# B&R Automation Studio project Tmp_Explorer_V1
Automation Studio 6.7.1.4; technology packages: mappServices 6.7.1, mappView 6.7.0, OpcUaCs 6.7.0

## Configuration X20CPU

CPU X20CP3687X, AutomationRuntime 6.7.8, Build 11.3.0, Safety 0.0

### Task classes (Cpu.sw)
```
Cyclic#8:
  FileExplor <- mappFileExplorer.FileExplorer.prg
  UsbDevice <- USBdevice.UsbDevice.prg
  NetDevice <- NETdevice.NetDevice.prg
Binaries: udbdef, mvLoader, TCData, ArSvcReg, mvConfig, arconfig, User, Role, iomap, asfw, ashwac, ashwd, sysconf, UaCsConfig, BRRole, Config, OpcUaMap
Libraries: FileIO, runtime, AsBrStr, AsUSB, standard, IecCheck, sys_lib, AsZip, AsICMP, astime, asieccon, UaCoalPrv, ArSsl, UaCoal, UaCore, MpServer, MpFile, MpBase
```

### Hardware
```
X20CP3687X : X20CP3687X v1.9.0.0
  Connector IF2:
    ActivateDevice = 1
    ActivateSnmp = 2
  Connector IF3:
    DNAConfiguration = manual
    CycleTime = 2000
  ConfigurationID = Tmp_Explorer_V1_X20CPU
  UserPartitionSize = 200
  VolatileGlobalPvSize = 200000
  EnableDebugger = 1
  FileDevice1
  FileDeviceName1 = USER
  FileDevicePath1 = USER_PATH
  ActivateFtpServer = 1
  FtpUser1
  FtpUsername1 = admin
  FtpUserPassword1 = 63faJ9mPKpD1G9ieIVwnNiGLd8KDZIbzebN9VYfcRfQ=  // admin
  FtpUserSalt1 = HY8+Pzqd
  FTPAccessRight1 = 0
  ActivateWebServer = 1
  ActivateSdm = 1
```

### Config.mpfilemanager - X20CP3687X/mappServices/Config.mpfilemanager
```
Element FileManagement (Type=mpfilemanager)
  mapp.Gen:
    Enable = TRUE
    EnableCockpit = TRUE
    Audit = TRUE
    Parent
  FileManager:
    USB = 0
    Devices:
      0:
        DeviceName = USER
        Text = USER
    Access:
      0:
        Folder = *
        Roles:
          0:
            Role = Everyone
            Rights:
              Visible = TRUE
              FolderRead = TRUE
              FileRead = TRUE
              FileEdit = TRUE
              FolderEdit = TRUE
          1:
            Role = Administrator
            Rights:
              Visible = TRUE
              FolderRead = TRUE
              FileRead = TRUE
              FileEdit = TRUE
              FolderEdit = TRUE
```

## Logical view

Binary libraries used (declarations not repeated): operator, runtime, astime, AsIecCon, FileIO, AsBrStr, AsUSB, standard, IecCheck, sys_lib, AsZip, AsICMP, MpServer 6.7.0, MpFile 6.7.1, MpBase

### compile_flags.txt
```
# This file is auto-generated by ASX. Do not edit manually, as changes may be overwritten.
# If you need to manually edit this file and prevent automatic updates, add "# MANUAL EDIT" to the first line.
-I
C:\Program Files (x86)\BrAutomation\AS6\AS\gnuinst\V11.3.0\6.0\i686-elf\include\c++\11.3.0
-I
C:\Program Files (x86)\BrAutomation\AS6\AS\gnuinst\V11.3.0\6.0\i686-elf\include\c++\11.3.0\i686-elf
-I
C:\Program Files (x86)\BrAutomation\AS6\AS\gnuinst\V11.3.0\6.0\i686-elf\include\c++\11.3.0\backward
-I
C:\Program Files (x86)\BrAutomation\AS6\AS\gnuinst\V11.3.0\6.0\lib\gcc\i686-elf\11.3.0\include
-I
C:\Program Files (x86)\BrAutomation\AS6\AS\gnuinst\V11.3.0\6.0\lib\gcc\i686-elf\11.3.0\include-fixed
-I
C:\Program Files (x86)\BrAutomation\AS6\AS\gnuinst\V11.3.0\6.0\i686-elf\include
-I
c:\Projects\Samples\mapp\mappExplorer\Temp\Includes
-trigraphs
-fno-asm
-D
_DEFAULT_INCLUDES
-D
_SG4
--target=i686-elf
-fPIC
-Wall
```

### ExplorerTypes.typ
```iecst
TYPE
	ClientInfoType : 	STRUCT
		userId : WSTRING[80];
		isValid : BOOL;
		ipAddress : WSTRING[15];
		languageId : WSTRING[2];
		screenResolution : WSTRING[32];
		slotId : SINT;
	END_STRUCT;
	expSTATE :
		( (*Explorer state machine*)
		EXP_WAIT,
		EXP_READ_DIR,
		EXP_READ_DIR_1,
		EXP_READ_DIR_2,
		EXP_READ_DIR_3,
		EXP_READ_DIR_4,
		EXP_DIR_CHANGE,
		EXP_COPY_ALL,
		EXP_FILE_COPY,
		EXP_FILE_DELETE,
		EXP_FILE_RENAME,
		EXP_FILE_DUPLICATE,
		EXP_FILE_VIEW,
		EXP_FILE_DOWNLOAD,
		EXP_FILE_DOWNLOAD_1,
		EXP_FILE_DOWNLOAD_DIR,
		EXP_FILE_UPLOAD,
		EXP_FILE_UPLOAD_1,
		EXP_DIR_COPY,
		EXP_DIR_CREATE,
		EXP_DIR_DELETE,
		EXP_DIR_RENAME,
		EXP_OVERWRITE_1,
		EXP_OVERWRITE_2
		);
	expERR : 	STRUCT  (*Sub structure error*)
		text : STRING[150]; (* Error text *)
		state : expSTATE; (* Error step *)
	END_STRUCT;
	expCMD : 	STRUCT  (*Sub structure commands*)
		refresh : BOOL; (*Read directory and file names from devices *)
		dir_change : BOOL; (*Change current directory *)
		dir_create : BOOL; (*Create a new directory *)
		copy : BOOL; (*Copy selected item from device a TO device b *)
		copy_all : BOOL; (*Copy all items from device a TO device b	*)
		view_file : BOOL; (*View selected file in mappView*)
		delete : BOOL; (*Delete selected file *)
		rename : BOOL; (*Rename selected file*)
		duplicate : BOOL; (*Duplicate selected file*)
		download : BOOL; (*Download selected file*)
		upload : BOOL; (*Upload file to target*)
	END_STRUCT;
	expPAR : 	STRUCT  (*Sub structure parameters*)
		device_active : STRING[40]; (*Active device name *)
		device_list : ARRAY[0..6]OF STRING[40]; (*List of all devices*)
		item_filter : STRING[EXPL_ITEM_LENGTH]; (*Only show files with this extension	*)
		new_name : STRING[EXPL_ITEM_LENGTH]; (*Name for for directory create and rename*)
		dir_path : STRING[EXPL_DIR_PATH_LENGTH]; (*Current directory path	*)
	END_STRUCT;
	expDAT : 	STRUCT  (*Sub structure data*)
		item_list : ARRAY[0..EXPL_LIST_NUM]OF STRING[EXPL_ITEM_LENGTH]; (*List with file names	*)
		item_size : ARRAY[0..EXPL_LIST_NUM]OF STRING[EXPL_SIZE_LENGTH]; (*List with file sizes*)
		item_num : UINT; (*Number of files	 displayed*)
		device_free : UINT; (*Free memory on device in MB*)
		device_size : UINT; (*Total memory size of device in MB*)
	END_STRUCT;
	expVIS : 	STRUCT  (*Sub structure visualization*)
		item_selected : UINT; (*Current selected file *)
		enable_button_set_1 : BOOL; (*Enable or disable buttons copy and delete*)
		enable_button_set_2 : BOOL; (*Enable or disable buttons refresh and create*)
		view_file_path : STRING[EXPL_DIR_PATH_LENGTH]; (*Full path for viewing file*)
		view_file : BOOL; (*Show message box on error*)
		download_execute : BOOL; (*Start downloading file*)
		file_status : DINT; (*Status of download and upload*)
		upload_execute : BOOL; (*Start uploading file*)
		file_full_path : STRING[EXPL_DIR_PATH_LENGTH]; (*File upload and download url*)
		overwrite_request : BOOL; (*Show message box to overwrite file*)
		overwrite_response : USINT; (*Response from message box overwrite file*)
		reload_upload : BOOL; (*Reload upload button*)
		double_click_event : USINT; (*Helper variable for double click in item list*)
		device_list : ARRAY[0..6]OF STRING[80]; (* Device name *)
	END_STRUCT;
	expMAIN : 	STRUCT  (*Main explorer structure*)
		CMD : ARRAY[0..1]OF expCMD; (* Command structure *)
		PAR : ARRAY[0..1]OF expPAR; (* Parameter structure *)
		DAT : ARRAY[0..1]OF expDAT; (*Data structure*)
		VIS : ARRAY[0..1]OF expVIS; (*Visualization structure*)
		ERR : expERR; (* Error structure *)
		status_no : DINT; (*Shows the status as number*)
		status_text : STRING[50]; (*Shows the status as text*)
	END_STRUCT;
END_TYPE
```

### ExplorerVariables.var
```iecst
VAR CONSTANT
	EXPL_DIR_PATH_LENGTH : UINT := 200; (*Maximum length for the complete path *)
	EXPL_LIST_NUM : UINT := 100; (*Maximum number if files and folders that can be listed *)
	EXPL_ITEM_LENGTH : USINT := 50; (*Maximum length for a file or folder name *)
	EXPL_SIZE_LENGTH : USINT := 15; (*Maximum length for a file or folder size*)
	EXPL_DEVICE_LIST : ARRAY[0..6] OF STRING[40] := ['USER','USB_DEVICE1','USB_DEVICE2','USB_DEVICE3','NET_DEVICE','','']; (*List of predefined devices *)
END_VAR
VAR
	EXPL_VIEW_FILTER : ARRAY[0..9] OF STRING[5] := ['csv','xml','txt','bmp','jpg',5('')]; (*Files extensions than can be used with the view command*)
	EXPL : expMAIN; (*Explorer main structure*)
END_VAR
```

### Program Logical/mappFileExplorer/FileExplorer (IEC)

#### Variables.var
```iecst
(*Local constants*)
VAR CONSTANT
	OK : USINT := 0; (*Status OK *)
	FILTER_AUTO_REFRESH : BOOL := TRUE; (*Auto refresh when filter changes *)
	COPY_AUTO_SELECT : USINT := 1; (*Select target item after copying *)
	COPY_AUTO_REFRESH : USINT := 1; (*Refresh items after copying *)
END_VAR
(*Local Variables*)
VAR
	side : BOOL := FALSE; (*Current side *)
	step : expSTATE := (0); (*Main step index *)
	animation : USINT := 0; (*Animation for working status	*)
	do_select : USINT := 0; (*Select item after copying *)
	old_filter : ARRAY[0..1] OF STRING[EXPL_ITEM_LENGTH]; (*Track filter change *)
	has_oversized_items : BOOL;
	tmp_str1 : STRING[EXPL_DIR_PATH_LENGTH]; (* Temporary STRING variable *)
	tmp_str2 : STRING[EXPL_DIR_PATH_LENGTH]; (* Temporary STRING variable *)
	tmp_str3 : STRING[EXPL_DIR_PATH_LENGTH]; (* Temporary STRING variable *)
	tmp_str4 : STRING[EXPL_DIR_PATH_LENGTH]; (* Temporary STRING variable *)
	lx : UDINT := 0; (* Index	*)
	ly : UINT;
	double_click_timer : TON_10ms;
	device_active_old : ARRAY[0..1] OF STRING[40];
	dir_path : STRING[EXPL_DIR_PATH_LENGTH];
	device_active : STRING[40];
	item_name : STRING[EXPL_DIR_PATH_LENGTH];
	duplicate_index : UDINT;
	duplicate_dot_pos : DINT;
	duplicate_suffix_pos : DINT;
	duplicate_suffix_valid : BOOL;
	duplicate_base_name : STRING[EXPL_ITEM_LENGTH];
	duplicate_extension : STRING[EXPL_ITEM_LENGTH];
	duplicate_suffix_text : STRING[EXPL_ITEM_LENGTH];
END_VAR
(*Local function calls*)
VAR
	DInfo : DirInfo;
	DOpen : DirOpen;
	DRead : DirReadEx;
	DClose : DirClose;
	FCopy : FileCopy;
	FDelete : FileDelete;
	FRename : FileRename;
	DCopy : DirCopy;
	DCreate : DirCreate;
	DDelete : DirDeleteEx;
	DRename : DirRename;
	DMemInfo : DevMemInfo;
	DevLink_0 : DevLink;
	lDirReadData : fiDIR_READ_EX_DATA;
	zipArchive_0 : zipArchive;
END_VAR
(*Local constants*)
VAR CONSTANT
	NONE : USINT := 0;
	YES : USINT := 1;
	NO : USINT := 2;
	ERR_EMPTY_ITEM : UINT := 50000; (*Selected item name is empty	*)
	ERR_INVALID_ITEM_NAME : UINT := 50001; (*This is not a valid item name*)
	ERR_DEVICE_UNDEFINED : UINT := 50010; (*Device is not defined*)
	ERR_MAX_FILES_REACHED : UINT := 50100; (*Maximum number of files reached*)
	ERR_NAME_EXCEEDS_MAX : UINT := 50200; (*File name exceeds maximum length*)
	ERR_DIR_EXCEEDS_MAX : UINT := 50201; (*Directory name exceeds maximum length*)
	ERR_PATH_EXCEEDS_MAX : UINT := 50202; (*Directory path exceeds maximum length*)
	ERR_PATH_CRITICAL : UINT := 50203; (*Directory path critical error*)
	ERR_PATH_RECURSIVE : UINT := 50204; (*Can not copy directory into itself*)
	ERR_DIR_DOWNLOAD_INVALID : UINT := 50331; (*This is not a valid directory for downloading*)
END_VAR
```

#### LocalFunctions.fun
```iecst
FUNCTION ReplaceString : BOOL
	VAR_INPUT
		dataSTR : UDINT;
		searchSTR : UDINT;
		replaceSTR : UDINT;
		first : BOOL;
	END_VAR
	VAR
		idx : UDINT;
	END_VAR
END_FUNCTION

FUNCTION IsInstr : BOOL
	VAR_INPUT
		string1 : UDINT;
		string2 : UDINT;
	END_VAR
	VAR
		idx : UDINT;
	END_VAR
END_FUNCTION

FUNCTION FindInMem : DINT
	VAR_INPUT
		data1 : UDINT;
		len1 : UDINT;
		data2 : UDINT;
		len2 : UDINT;
		direction : BOOL;
	END_VAR
	VAR
		idx : UDINT;
	END_VAR
END_FUNCTION

{REDUND_ERROR} FUNCTION CreateError : expSTATE (*TODO: Add your comment here*) (*$GROUP=User,$CAT=User,$GROUPICON=User.png,$CATICON=User.png*)
	VAR_INPUT
		nr : DINT;
		side : BOOL;
		step : expSTATE;
		text : STRING[150];
		EXPL : REFERENCE TO expMAIN;
	END_VAR
END_FUNCTION

FUNCTION InsertRecName : BOOL
	VAR_INPUT
		EXPL : REFERENCE TO expMAIN;
		new_name : STRING[EXPL_ITEM_LENGTH];
		size : STRING[15];
		side : BOOL;
	END_VAR
	VAR
		idx : DINT;
		idy : DINT;
		lSort : DINT;
	END_VAR
END_FUNCTION

FUNCTION WorkingStatus : USINT
	VAR_INPUT
		EXPL : REFERENCE TO expMAIN;
		str : UDINT;
		animation : USINT;
	END_VAR
END_FUNCTION

FUNCTION CreateCompletePath : BOOL
	VAR_INPUT
		path : STRING[EXPL_DIR_PATH_LENGTH];
		target : STRING[EXPL_ITEM_LENGTH];
		return_path : UDINT;
	END_VAR
	VAR
		tmp : STRING[EXPL_ITEM_LENGTH];
	END_VAR
END_FUNCTION

FUNCTION String2DataProvider : BOOL
	VAR_INPUT
		SourceString : UDINT;
		TargetString : UDINT;
	END_VAR
END_FUNCTION
```

#### LocalFunctions.st
```iecst
//******************************************************************************************************
// Create mappView data provider string
//******************************************************************************************************
FUNCTION String2DataProvider
	brsstrcpy(TargetString, ADR('{"value":"'));
	brsstrcat(TargetString, SourceString);
	brsstrcat(TargetString, ADR('","text":"'));
	brsstrcat(TargetString, SourceString);
	brsstrcat(TargetString, ADR('"}'));
	String2DataProvider := TRUE;
END_FUNCTION

//******************************************************************************************************
// Raise error function
//******************************************************************************************************
FUNCTION CreateError
	// Generate for known errors
	IF (nr = fiERR_NOT_ENOUGH_FREEMEM) THEN
		EXPL.ERR.text := 'not enough memory available on the target device';
	ELSIF (nr = fiERR_FILE_DEVICE) THEN
		EXPL.ERR.text := 'device is not connected';
	ELSIF (nr = fiERR_INVALID_PATH) THEN
		EXPL.ERR.text := 'directory is too long, does not exist or has invalid characters';
	ELSIF (nr = fiERR_DIR_NOT_EXIST) THEN
		EXPL.ERR.text := 'directory does not exist';
	ELSIF (nr = fiERR_FILE_DEVICE) THEN
		EXPL.ERR.text := 'directory path does not exist';
	ELSIF (nr = fiERR_DIR_ALREADY_EXIST) THEN
		EXPL.ERR.text := 'directory or file already exists';
	ELSIF (nr = fiERR_EXIST) THEN
		EXPL.ERR.text := 'directory or file already exists';
	ELSE
		EXPL.ERR.text := text;
	END_IF
	// Convert to error structure
	IF (side = 0) THEN
		brsstrcat(ADR(EXPL.ERR.text), ADR(' on side a'));
	ELSE
		brsstrcat(ADR(EXPL.ERR.text), ADR(' on side b'));
	END_IF
	EXPL.status_no 	:= nr;
	EXPL.ERR.state 	:= step;
	// When error occurs in dir read call dir close before reporting error
	IF (step = EXP_READ_DIR_2) THEN
		CreateError := EXP_READ_DIR_3;
	ELSE
		// Reset all commands
		brsmemset(ADR(EXPL.CMD[side]), 0, SIZEOF(EXPL.CMD[side]));
		brsmemset(ADR(EXPL.CMD[NOT side]), 0, SIZEOF(EXPL.CMD[NOT side]));
		CreateError := EXP_WAIT;
	END_IF
END_FUNCTION

//******************************************************************************************************
// Create complete path string
//******************************************************************************************************
FUNCTION CreateCompletePath
	brsmemset(ADR(tmp), 0, EXPL_ITEM_LENGTH);
	brsstrcpy(return_path, ADR(path));

	// ------------------------------------------------------------------------------------------------
	// Filter directory name
	IF(brsmemcmp(ADR(target), ADR('(DIR)'), 5) = 0) THEN
		brsmemcpy(ADR(tmp), ADR(target)+5, brsstrlen(ADR(target))-5);
	ELSE
		brsstrcpy(ADR(tmp), ADR(target));
	END_IF

	// ------------------------------------------------------------------------------------------------
	// Create directory path
	IF(path = '/') THEN
		brsstrcpy(return_path, ADR(tmp));
	ELSE
		brsstrcat(return_path, ADR('/'));
		brsstrcat(return_path, ADR(tmp));
	END_IF
	//	brsstrcat(return_path, ADR('/'));

	CreateCompletePath := FALSE;
END_FUNCTION

//******************************************************************************************************
// Working status
//******************************************************************************************************
FUNCTION WorkingStatus
	animation := animation+1;

	IF (animation = 80) THEN
		animation := 0;
	END_IF

	brsmemset(ADR(EXPL.status_text), 0, SIZEOF(EXPL.status_text));
	brsstrcpy(ADR(EXPL.status_text), str);
	CASE(animation) OF
		0..19	: brsstrcat(ADR(EXPL.status_text), ADR('/'));
		20..39	: brsstrcat(ADR(EXPL.status_text), ADR('-'));
		40..59	: brsstrcat(ADR(EXPL.status_text), ADR('\'));
		60..79	: brsstrcat(ADR(EXPL.status_text), ADR('|'));
	END_CASE;
	WorkingStatus := animation;
END_FUNCTION

//******************************************************************************************************
// Fill new folder or directory name
//******************************************************************************************************
FUNCTION InsertRecName
	// Set up start values for iteration
	IF (EXPL.DAT[side].item_num <> 0) THEN
		idy := EXPL.DAT[side].item_num - 1;
	END_IF
	idx := idy;

	// Start iteration	search
	WHILE (idy > 1) DO
		// Check current entry
		lSort := brsstrcmp(ADR(new_name), ADR(EXPL.DAT[side].item_list[idy]));
		// Solve new search range
		IF (idy MOD 2 = 0) THEN
			idy := idy / 2;
		ELSE
			idy := idy / 2 + 1;
		END_IF
		// New range is lower or higher than current
		IF (lSort > 0) THEN
			idx := idx + idy;
			IF (idx > UINT_TO_INT(EXPL.DAT[side].item_num)) THEN
				idx := EXPL.DAT[side].item_num;
			END_IF
		ELSE
			idx := idx - idy;
			IF (idx < 1) THEN
				idx := 1;
			END_IF
		END_IF
	END_WHILE;

	// New entry is this, next or previous
	lSort := brsstrcmp(ADR(new_name), ADR(EXPL.DAT[side].item_list[idx]));
	IF (lSort > 0 AND idx <> UINT_TO_INT(EXPL.DAT[side].item_num)) THEN
		idx := idx +1;
	ELSIF (idx > 0) THEN
		lSort := brsstrcmp(ADR(new_name), ADR(EXPL.DAT[side].item_list[idx-1]));
		IF (lSort < 0) THEN
			idx := idx - 1;
		END_IF
	END_IF

	// Force ".." at beginning of list
	IF (idx = 0 AND EXPL.DAT[side].item_list[0] = '..') THEN
		idx := idx + 1;
	END_IF
	// Move all data entrys backwards and fill in new entry
	IF(idx < EXPL_LIST_NUM) THEN
		brsmemmove(ADR(EXPL.DAT[side].item_list[idx+1]),ADR(EXPL.DAT[side].item_list[idx]), (EXPL.DAT[side].item_num - idx) * SIZEOF(EXPL.DAT[side].item_list[0]));
		brsmemmove(ADR(EXPL.DAT[side].item_size[idx+1]),ADR(EXPL.DAT[side].item_size[idx]), (EXPL.DAT[side].item_num - idx) * SIZEOF(EXPL.DAT[side].item_size[0]));
	END_IF
	brsstrcpy(ADR(EXPL.DAT[side].item_list[idx]), ADR(new_name));
	// Create data structure for vis size list
	brsstrcpy(ADR(EXPL.DAT[side].item_size[idx]), ADR(size));

	InsertRecName := TRUE;
END_FUNCTION

//******************************************************************************************************
// Is second string in first string
//******************************************************************************************************
FUNCTION IsInstr
	IF (brsstrlen(string1) > brsstrlen(string2)) THEN
		FOR idx:=0 TO brsstrlen(string1) - brsstrlen(string2) DO
			IF (brsmemcmp(string1 + idx, string2, brsstrlen(string2)) = 0) THEN
				IsInstr := TRUE;
				EXIT;
			END_IF
		END_FOR;
	END_IF
END_FUNCTION

//******************************************************************************************************
// Find second data in first data
//******************************************************************************************************
FUNCTION FindInMem
	FindInMem := -1;
	IF (len1 > len2) THEN
		IF(direction) THEN
			idx := len1 - len2;
			WHILE(idx > 0) DO
				IF (brsmemcmp(data1 + idx, data2, len2) = 0) THEN
					FindInMem := idx;
					EXIT;
				END_IF
				idx := idx - 1;
			END_WHILE;
		ELSE
			FOR idx:=0 TO len1 - len2 DO
				IF (brsmemcmp(data1 + idx, data2, len2) = 0) THEN
					FindInMem := idx;
					EXIT;
				END_IF
			END_FOR;
		END_IF
	END_IF
END_FUNCTION

//******************************************************************************************************
// Find and replace string
//******************************************************************************************************
FUNCTION ReplaceString
	IF (brsstrlen(dataSTR) >= brsstrlen(searchSTR)) THEN
		FOR idx:=0 TO brsstrlen(dataSTR) - brsstrlen(searchSTR) DO
			IF (brsmemcmp(dataSTR + idx, searchSTR, brsstrlen(searchSTR)) = 0) THEN
				// Move data around
				brsmemmove(dataSTR + idx + brsstrlen(replaceSTR), dataSTR + idx + brsstrlen(searchSTR), brsstrlen(dataSTR) - brsstrlen(searchSTR) + 1);
				brsmemcpy(dataSTR + idx, replaceSTR, brsstrlen(replaceSTR));
				// Set found flag and exit if only one hit is needed
				ReplaceString := TRUE;
				IF(first) THEN
					EXIT;
				END_IF
				// Correct index for next search
				IF(brsstrlen(replaceSTR) > 0) THEN
					idx := idx + brsstrlen(replaceSTR);
				END_IF
				idx := idx - 1;
				// Exit if no data is left
				IF (brsstrlen(dataSTR) = 0 OR brsstrlen(dataSTR) < brsstrlen(searchSTR)) THEN
					EXIT;
				END_IF
			END_IF
		END_FOR;
	END_IF
END_FUNCTION
```

#### Main.st
```iecst
// ----------------------------------------------------------------------------------------
//	Function: mappView explorer
// ----------------------------------------------------------------------------------------

PROGRAM _INIT
	// ----------------------------------------------------------------------------------------
	// Copy pre-configured devices into list
	brsmemcpy(ADR(EXPL.PAR[0].device_list), ADR(EXPL_DEVICE_LIST), SIZEOF(EXPL_DEVICE_LIST));
	brsmemcpy(ADR(EXPL.PAR[1].device_list), ADR(EXPL_DEVICE_LIST), SIZEOF(EXPL_DEVICE_LIST));
	brsstrcpy(ADR(EXPL.PAR[0].device_active), ADR(EXPL.PAR[0].device_list[0]));
	brsstrcpy(ADR(EXPL.PAR[1].device_active), ADR(EXPL.PAR[1].device_list[0]));

	// ----------------------------------------------------------------------------------------
	// Connect to user device for temporary files used with download all
	REPEAT
		DevLink_0.enable := 1;
		DevLink_0.pDevice := ADR('TMP_USER');
		DevLink_0.pParam := ADR('/DEVICE=F:');
		DevLink_0;
		UNTIL DevLink_0.status <> ERR_FUB_BUSY
	END_REPEAT;
END_PROGRAM

PROGRAM _CYCLIC

	// ------------------------------------------------------------------------------------------------
	// Set switches for HMI, these buttons are enabled if there is at least one file or directory
	IF(EXPL.DAT[side].item_num > 0) THEN
		EXPL.VIS[side].enable_button_set_1 := TRUE;
	ELSE
		EXPL.VIS[side].enable_button_set_1 := FALSE;
	END_IF

	// ------------------------------------------------------------------------------------------------
	// Generate device name list for drop down box
	brsmemset(ADR(EXPL.VIS[side].device_list), 0, SIZEOF(EXPL.VIS[side].device_list));
	FOR lx := 0 TO SIZEOF(EXPL.VIS[side].device_list)/SIZEOF(EXPL.VIS[side].device_list[0]) - 1 DO
		IF (EXPL.PAR[side].device_list[lx] <> '') THEN
			String2DataProvider(ADR(EXPL.PAR[side].device_list[lx]), ADR(EXPL.VIS[side].device_list[lx]));
		END_IF
	END_FOR;

	// ------------------------------------------------------------------------------------------------
	// Handle double click for directory change and file view
	IF(EXPL.VIS[side].double_click_event > 0) THEN
		double_click_timer.PT := 50;
		double_click_timer.IN := TRUE;
		double_click_timer();
		IF(EXPL.VIS[side].double_click_event > 1) THEN
			double_click_timer.IN := FALSE;
			double_click_timer();
			EXPL.VIS[side].double_click_event := 0;
			IF(brsmemcmp(ADR(EXPL.DAT[side].item_list[EXPL.VIS[side].item_selected]), ADR('(DIR)'), 5) = 0 OR EXPL.DAT[side].item_list[EXPL.VIS[side].item_selected] = '..') THEN
				EXPL.CMD[side].dir_change := TRUE;
			ELSE
				EXPL.CMD[side].view_file := TRUE;
			END_IF
		END_IF
	END_IF
	IF(double_click_timer.Q) THEN
		double_click_timer.IN := FALSE;
		double_click_timer();
		IF(EXPL.VIS[side].double_click_event > 0) THEN
			EXPL.VIS[side].double_click_event := EXPL.VIS[side].double_click_event - 1;
		END_IF
	END_IF

	//--------------------------------------------------------------------------------------------------
	// Check if parameters are valid
	IF (EXPL.PAR[side].device_active = '') THEN
		step := CreateError(ERR_DEVICE_UNDEFINED, side, step, 'device is not defined', ADR(EXPL));
		RETURN;
	END_IF
	IF (brsstrlen(ADR(EXPL.PAR[side].dir_path)) >= EXPL_DIR_PATH_LENGTH) THEN
		step := CreateError(ERR_PATH_CRITICAL, side, step, 'directory path critical error', ADR(EXPL));
		RETURN;
	END_IF

	// ------------------------------------------------------------------------------------------------
	// Track filter change
	IF (FILTER_AUTO_REFRESH AND brsstrcmp(ADR(old_filter[side]), ADR(EXPL.PAR[side].item_filter)) <> 0) THEN
		brsstrcpy(ADR(old_filter[side]), ADR(EXPL.PAR[side].item_filter));
		EXPL.CMD[side].refresh	:= TRUE;
	END_IF

	// ------------------------------------------------------------------------------------------------
	// Track device name change
	IF(device_active_old[side] <> EXPL.PAR[side].device_active) THEN
		EXPL.PAR[side].dir_path := '';
		EXPL.CMD[side].refresh	:= TRUE;
	END_IF
	device_active_old[side] := EXPL.PAR[side].device_active;

	// ------------------------------------------------------------------------------------------------
	// Stop here if no command is set
	IF (EXPL.CMD[side].refresh = FALSE AND EXPL.CMD[side].dir_change = FALSE AND EXPL.CMD[side].dir_create = FALSE AND EXPL.CMD[side].copy = FALSE AND EXPL.CMD[side].copy_all = FALSE AND EXPL.CMD[side].delete = FALSE AND EXPL.CMD[side].rename = FALSE AND EXPL.CMD[side].duplicate = FALSE AND EXPL.CMD[side].view_file = FALSE AND EXPL.CMD[side].download = FALSE AND EXPL.CMD[side].upload = FALSE) THEN
		// --------------------------------------------------------------------------------------------
		// Show current state
		EXPL.status_text := 'Waiting...';
		// --------------------------------------------------------------------------------------------
		// If selection is out of range set it to maximum
		IF ((EXPL.VIS[side].item_selected > EXPL.DAT[side].item_num - 1) AND (EXPL.DAT[side].item_num <> 0)) THEN
			EXPL.VIS[side].item_selected := EXPL.DAT[side].item_num - 1;
		END_IF
		side := NOT side;
		// Enable buttons when command is active
		EXPL.VIS[0].enable_button_set_2 := TRUE;
		EXPL.VIS[1].enable_button_set_2 := TRUE;
		// Reset busy status
		IF (EXPL.ERR.state = 0) AND (EXPL.status_no = ERR_FUB_BUSY) THEN
			EXPL.status_no := 0;
		END_IF
		RETURN;
	END_IF

	// Disable buttons when command is active
	EXPL.VIS[0].enable_button_set_1 := FALSE;
	EXPL.VIS[1].enable_button_set_1 := FALSE;
	EXPL.VIS[0].enable_button_set_2 := FALSE;
	EXPL.VIS[1].enable_button_set_2 := FALSE;

	// Clear errors on new command
	brsmemset(ADR(EXPL.ERR), 0, SIZEOF(EXPL.ERR));

	//**************************************************************************************************
	// Cyclic Part
	//**************************************************************************************************
	CASE step OF
		//**********************************************************************************************
		// Wait for command
		//**********************************************************************************************
		EXP_WAIT:
			// ----------------------------------------------------------------------------------------
			// Refresh direcrory information
			IF (EXPL.CMD[side].refresh = TRUE) THEN
				step := EXP_READ_DIR;
			END_IF
			// ----------------------------------------------------------------------------------------
			// Change active directory
			IF (EXPL.CMD[side].dir_change = TRUE) THEN
				// ------------------------------------------------------------------------------------
				// Check if directory name is empty
				IF (EXPL.DAT[side].item_list[EXPL.VIS[side].item_selected] = '') THEN
					step := CreateError(ERR_EMPTY_ITEM, side, step, 'directory name is empty', ADR(EXPL));
					// Check if directory name is valid
				ELSIF((brsmemcmp(ADR(EXPL.DAT[side].item_list[EXPL.VIS[side].item_selected]), ADR('(DIR)'), 5) <> 0) AND (EXPL.DAT[side].item_list[EXPL.VIS[side].item_selected] <> '..'))  THEN
					step := CreateError(ERR_INVALID_ITEM_NAME, side, step, 'this is not a valid directory name', ADR(EXPL));
					// Check if new directory name fits into string
				ELSIF(brsstrlen(ADR(EXPL.DAT[side].item_list[EXPL.VIS[side].item_selected])) - 5 + brsstrlen(ADR(EXPL.PAR[side].dir_path)) + 1 >= EXPL_DIR_PATH_LENGTH) THEN
					step := CreateError(ERR_PATH_EXCEEDS_MAX, side, step, 'directory path exceeds maximum length', ADR(EXPL));
				ELSE
					step := EXP_DIR_CHANGE;
				END_IF
			END_IF
			// ----------------------------------------------------------------------------------------
			// Create a new directory
			IF (EXPL.CMD[side].dir_create = TRUE) THEN
				// ------------------------------------------------------------------------------------
				// Check if new directory name is empty
				IF (EXPL.PAR[side].new_name = '') THEN
					step := CreateError(ERR_EMPTY_ITEM, side, step, 'directory name is empty', ADR(EXPL));
					// Check if new directory name fits into path string
				ELSIF(brsstrlen(ADR(EXPL.PAR[side].new_name)) + brsstrlen(ADR(EXPL.PAR[side].dir_path)) + 1 >= EXPL_DIR_PATH_LENGTH) THEN
					step := CreateError(ERR_PATH_EXCEEDS_MAX, side, step, 'directory path name exceeds maximum length', ADR(EXPL));
					// Check if new directory name fits into directory name string
				ELSIF(brsstrlen(ADR(EXPL.PAR[side].new_name)) + 5 >= EXPL_ITEM_LENGTH) THEN
					step := CreateError(ERR_DIR_EXCEEDS_MAX, side, step, 'directory name exceeds maximum length', ADR(EXPL));
				ELSE
					step := EXP_DIR_CREATE;
				END_IF
			END_IF
			// ----------------------------------------------------------------------------------------
			// Copy one file
			IF (EXPL.CMD[side].copy = TRUE) THEN
				// ------------------------------------------------------------------------------------
				// Make sure that user chooses a valid item
				IF (EXPL.DAT[side].item_list[EXPL.VIS[side].item_selected] = '..') THEN
					step := CreateError(ERR_INVALID_ITEM_NAME, side, step, 'this is not a valid item name', ADR(EXPL));
				ELSE
					item_name := EXPL.DAT[side].item_list[EXPL.VIS[side].item_selected];
					step := EXP_OVERWRITE_1;
				END_IF
			END_IF
			// ----------------------------------------------------------------------------------------
			// Copy all files and folders in this directory
			IF (EXPL.CMD[side].copy_all = TRUE) THEN
				step := EXP_COPY_ALL;
			END_IF
			// ----------------------------------------------------------------------------------------
			// View selected file
			IF (EXPL.CMD[side].view_file = TRUE) THEN
				step := EXP_FILE_VIEW;
			END_IF
			// ----------------------------------------------------------------------------------------
			// Download selected file or directory
			IF (EXPL.CMD[side].download = TRUE) THEN
				EXPL.VIS[side].file_full_path := '';
				item_name := EXPL.DAT[side].item_list[EXPL.VIS[side].item_selected];
				// Make sure selected entry is valid
				IF(brsmemcmp(ADR(item_name), ADR('..'), 2) <> 0) THEN
					// Check if selected item is a single file
					IF(brsmemcmp(ADR(item_name), ADR('(DIR)'), 5) <> 0) THEN
						device_active := EXPL.PAR[side].device_active;
						dir_path := EXPL.PAR[side].dir_path;
						step := EXP_FILE_DOWNLOAD;
						// Selected item is a directory
					ELSE
						ReplaceString(ADR(item_name), ADR('(DIR)'), ADR(''), TRUE);
						step := EXP_FILE_DOWNLOAD_DIR;
					END_IF
				ELSE
					step := CreateError(ERR_DIR_DOWNLOAD_INVALID, side, step, 'item is not a valid directory', ADR(EXPL));
				END_IF
			END_IF
			// ----------------------------------------------------------------------------------------
			// Upload a new file
			IF (EXPL.CMD[side].upload = TRUE) THEN
				EXPL.VIS[side].file_full_path := '';
				device_active := EXPL.PAR[side].device_active;
				dir_path := EXPL.PAR[side].dir_path;
				step := EXP_FILE_UPLOAD;
			END_IF
			// ----------------------------------------------------------------------------------------
			// Delete the selected file
			IF (EXPL.CMD[side].delete = 1) THEN
				// Check if directory name is empty
				IF (EXPL.DAT[side].item_list[EXPL.VIS[side].item_selected] = '')	THEN
					step := CreateError(ERR_EMPTY_ITEM, side, step, 'item name is empty', ADR(EXPL));
					// Check if new directory name fits into string
				ELSIF(brsstrlen(ADR(EXPL.DAT[side].item_list[EXPL.VIS[side].item_selected])) + brsstrlen(ADR(EXPL.PAR[side].dir_path)) + 1 >= EXPL_DIR_PATH_LENGTH + EXPL_ITEM_LENGTH) THEN
					step := CreateError(ERR_PATH_EXCEEDS_MAX, side, step, 'directory path exceeds maximum length', ADR(EXPL));
					// Make sure that a valid item was selected
				ELSIF(EXPL.DAT[side].item_list[EXPL.VIS[side].item_selected] = '..') THEN
					step := CreateError(ERR_INVALID_ITEM_NAME, side, step, 'this is not a valid item name', ADR(EXPL));
					// Delete a directory
				ELSIF(brsmemcmp(ADR(EXPL.DAT[side].item_list[EXPL.VIS[side].item_selected]), ADR('(DIR)'), 5) = 0)	THEN
					item_name := EXPL.DAT[side].item_list[EXPL.VIS[side].item_selected];
					step := EXP_DIR_DELETE;
					// Delete a file
				ELSE
					item_name := EXPL.DAT[side].item_list[EXPL.VIS[side].item_selected];
					step := EXP_FILE_DELETE;
				END_IF
			END_IF
			// ----------------------------------------------------------------------------------------
			// Rename file or directory
			IF (EXPL.CMD[side].rename = TRUE) THEN
				// ------------------------------------------------------------------------------------
				// Check if new name is empty
				IF (EXPL.PAR[side].new_name = '') THEN
					step := CreateError(ERR_EMPTY_ITEM, side, step, 'new name is empty', ADR(EXPL));
					// Make sure that a valid item was selected
				ELSIF (EXPL.DAT[side].item_list[EXPL.VIS[side].item_selected] = '..') THEN
					step := CreateError(ERR_INVALID_ITEM_NAME, side, step, 'this is not a valid item name', ADR(EXPL));
					// Check if new directory name exceeds maximum length
				ELSIF((brsmemcmp(ADR(EXPL.DAT[side].item_list[EXPL.VIS[side].item_selected]), ADR('(DIR)'), 5) = 0) AND (brsstrlen(ADR(EXPL.PAR[side].new_name)) + 5 >= EXPL_ITEM_LENGTH)) THEN
					step := CreateError(ERR_DIR_EXCEEDS_MAX, side, step, 'directory name exceeds maximum length', ADR(EXPL));
					// Check if new file name exceeds maximum length
				ELSIF (brsstrlen(ADR(EXPL.PAR[side].new_name)) >= EXPL_ITEM_LENGTH) THEN
					step := CreateError(ERR_NAME_EXCEEDS_MAX, side, step, 'file name exceeds maximum length', ADR(EXPL));
					// Rename a directory
				ELSIF(brsmemcmp(ADR(EXPL.DAT[side].item_list[EXPL.VIS[side].item_selected]), ADR('(DIR)'), 5) = 0)	THEN
					step := EXP_DIR_RENAME;
					// Rename a file
				ELSE
					step := EXP_FILE_RENAME;
				END_IF
			END_IF
			// ----------------------------------------------------------------------------------------
			// Duplicate selected file
			IF (EXPL.CMD[side].duplicate = TRUE) THEN
				// Make sure that a valid file was selected
				IF (EXPL.DAT[side].item_list[EXPL.VIS[side].item_selected] = '' OR EXPL.DAT[side].item_list[EXPL.VIS[side].item_selected] = '..') THEN
					step := CreateError(ERR_INVALID_ITEM_NAME, side, step, 'this is not a valid item name', ADR(EXPL));
				ELSIF (brsmemcmp(ADR(EXPL.DAT[side].item_list[EXPL.VIS[side].item_selected]), ADR('(DIR)'), 5) = 0) THEN
					step := CreateError(ERR_INVALID_ITEM_NAME, side, step, 'duplicate is only supported for files', ADR(EXPL));
					// Check if custom target name fits into path string
				ELSIF (EXPL.PAR[side].new_name <> '' AND brsstrlen(ADR(EXPL.PAR[side].new_name)) + brsstrlen(ADR(EXPL.PAR[side].dir_path)) + 1 >= EXPL_DIR_PATH_LENGTH) THEN
					step := CreateError(ERR_PATH_EXCEEDS_MAX, side, step, 'duplicate file path exceeds maximum length', ADR(EXPL));
				ELSE
					item_name := EXPL.DAT[side].item_list[EXPL.VIS[side].item_selected];
					duplicate_index := 0;
					step := EXP_FILE_DUPLICATE;
				END_IF
			END_IF

			// Set status
			EXPL.status_no := ERR_FUB_BUSY;

			//**********************************************************************************************
			// Read directory information
			//**********************************************************************************************
		EXP_READ_DIR:
			// Show current state
			animation := animation := WorkingStatus(ADR(EXPL), ADR('reading directory...'), animation);
			// ----------------------------------------------------------------------------------------
			// Clear all entrys
			brsmemset(ADR(EXPL.DAT[side]), 0, SIZEOF(EXPL.DAT[side]));
			EXPL.VIS[side].item_selected := 0;
			EXPL.DAT[side].item_num := 0;
			// ----------------------------------------------------------------------------------------
			// Add .. for directory up
			IF(EXPL.PAR[side].dir_path <> '/' AND EXPL.PAR[side].dir_path <> '') THEN
				EXPL.DAT[side].item_list[0] := '..';
				EXPL.DAT[side].item_num := 1;
			END_IF
			// ----------------------------------------------------------------------------------------
			// Set parameters and get device dir
			DInfo.enable 	:= TRUE;
			DInfo.pDevice	:= ADR(EXPL.PAR[side].device_active);
			DInfo.pPath 	:= ADR(EXPL.PAR[side].dir_path);
			DInfo();

			// ----------------------------------------------------------------------------------------
			// OK
			IF (DInfo.status = OK) THEN
				step := EXP_READ_DIR_1;
				// ----------------------------------------------------------------------------------------
				// Device is not available
			ELSIF (DInfo.status = fiERR_FILE_DEVICE) THEN
				EXPL.DAT[side].item_list[0] := 'not connected';
				step := CreateError(DInfo.status, side, step, 'not connected', ADR(EXPL));
				// ----------------------------------------------------------------------------------------
				// Device is not available
			ELSIF (DInfo.status = fiERR_DEVICE_MANAGER) THEN
				EXPL.DAT[side].item_list[0] := 'not connected';
				step := CreateError(DInfo.status, side, step, 'check device name and path', ADR(EXPL));
				// Error
			ELSIF (DInfo.status <> ERR_FUB_BUSY) THEN
				step := CreateError(DInfo.status, side, step, 'error dir info', ADR(EXPL));
			END_IF
			//**********************************************************************************************
			// Open directory
			//**********************************************************************************************
		EXP_READ_DIR_1:
			// Add current directory
			IF(EXPL.PAR[side].dir_path = '') THEN
				EXPL.PAR[side].dir_path := '/';
			END_IF
			DOpen.enable 	:= TRUE;
			DOpen.pDevice	:= ADR(EXPL.PAR[side].device_active);
			DOpen.pName 	:= ADR(EXPL.PAR[side].dir_path);
			DOpen();

			// ----------------------------------------------------------------------------------------
			// OK
			IF (DOpen.status = OK) THEN
				has_oversized_items := FALSE;
				step := EXP_READ_DIR_2;
				// Error
			ELSIF (DOpen.status <> ERR_FUB_BUSY) THEN
				step := CreateError(DOpen.status, side, step, 'error dir open', ADR(EXPL));
			END_IF;
			//**********************************************************************************************
			// Read file directory information
			//**********************************************************************************************
		EXP_READ_DIR_2:
			DRead.enable 	:= TRUE;
			DRead.ident		:= DOpen.ident;
			DRead.pData 	:= ADR(lDirReadData);
			DRead.data_len 	:= SIZEOF(lDirReadData);
			DRead();

			// ----------------------------------------------------------------------------------------
			// OK
			IF (DRead.status = OK) THEN
				// ------------------------------------------------------------------------------------
				// Verify that we still have space in list
				IF (EXPL.DAT[side].item_num < SIZEOF(EXPL.DAT[side].item_list)/SIZEOF(EXPL.DAT[side].item_list[0])) THEN
					// --------------------------------------------------------------------------------
					// Make sure file name contains filter
					IF (brsstrlen(ADR(EXPL.PAR[side].item_filter)) = 0 OR IsInstr(ADR(lDirReadData.Filename), ADR(EXPL.PAR[side].item_filter))) THEN
						brsmemset(ADR(tmp_str1), 0, SIZEOF(tmp_str1));
						// ----------------------------------------------------------------------------
						// Read file information
						IF (lDirReadData.Mode = fiFILE) THEN
							IF (brsstrlen(ADR(lDirReadData.Filename)) < EXPL_ITEM_LENGTH) THEN
								brsstrcpy(ADR(tmp_str1), ADR(lDirReadData.Filename));
								// --------------------------------------------------------------------
								// Generate file size
								IF (lDirReadData.Filelength > 1048576) THEN
									brsitoa(lDirReadData.Filelength/1048576, ADR(tmp_str2));
									brsstrcat(ADR(tmp_str2), ADR('M'));
								ELSIF (lDirReadData.Filelength > 1024) THEN
									brsitoa(lDirReadData.Filelength/1024, ADR(tmp_str2));
									brsstrcat(ADR(tmp_str2), ADR('K'));
								ELSE
									brsitoa(lDirReadData.Filelength, ADR(tmp_str2));
								END_IF
								InsertRecName(ADR(EXPL), tmp_str1, tmp_str2, side);
								EXPL.DAT[side].item_num := EXPL.DAT[side].item_num + 1;
							ELSE
								has_oversized_items := TRUE;
							END_IF
							// ----------------------------------------------------------------------------
							// Read directory information
						ELSIF (brsstrcmp(ADR(lDirReadData.Filename), ADR('.')) <> 0 AND brsstrcmp(ADR(lDirReadData.Filename), ADR('..')) <> 0 AND brsstrcmp(ADR(lDirReadData.Filename), ADR('System Volume Information')) <> 0) THEN
							IF (brsstrlen(ADR(lDirReadData.Filename)) < EXPL_ITEM_LENGTH-5) THEN
								// Copy directory name
								tmp_str1 := '(DIR)';
								brsstrcat(ADR(tmp_str1), ADR(lDirReadData.Filename));
								InsertRecName(ADR(EXPL), tmp_str1, '', side);
								EXPL.DAT[side].item_num := EXPL.DAT[side].item_num + 1;
							ELSE
								has_oversized_items := TRUE;
							END_IF
						END_IF
					END_IF
				ELSE
					step := CreateError(ERR_MAX_FILES_REACHED, side, step, 'maximum number of files reached', ADR(EXPL));
				END_IF
				// Last entry reached
			ELSIF (DRead.status = fiERR_NO_MORE_ENTRIES) THEN
				step := EXP_READ_DIR_3;
				// Error
			ELSIF (DRead.status <> ERR_FUB_BUSY) THEN
				step := CreateError(DRead.status, side, step, 'error dir read', ADR(EXPL));
			END_IF
			//**********************************************************************************************
			// Close directory information
			//**********************************************************************************************
		EXP_READ_DIR_3:
			DClose.enable 	:= TRUE;
			DClose.ident	:= DOpen.ident;
			DClose();

			// ----------------------------------------------------------------------------------------
			// OK
			IF (DClose.status = OK) THEN
				// Report error from dir read
				IF (DRead.status <> ERR_OK AND DRead.status <> fiERR_NO_MORE_ENTRIES) THEN
					step := CreateError(DRead.status, side, step, 'error dir read', ADR(EXPL));
				ELSE
					DClose.ident := 0;
					step := EXP_READ_DIR_4;
				END_IF
				// Error
			ELSIF (DClose.status <> ERR_FUB_BUSY) THEN
				step := CreateError(DClose.status, side, step, 'error dir close', ADR(EXPL));
			END_IF
			//**********************************************************************************************
			// Get device memory information
			//**********************************************************************************************
		EXP_READ_DIR_4:
				IF (NET.PAR.server_protocol = 'ftp' AND EXPL.PAR[side].device_active = 'NET_DEVICE') THEN
					DMemInfo(enable := FALSE);
					EXPL.DAT[side].device_free := 0;
					EXPL.DAT[side].device_size := 0;
				ELSE
					DMemInfo.enable 	:= TRUE;
					DMemInfo.pDevice	:= ADR(EXPL.PAR[side].device_active);
					DMemInfo();
					IF (DMemInfo.status = OK) THEN
						// Transfer device memory information
						EXPL.DAT[side].device_free := UDINT_TO_INT(DMemInfo.freemem/1048576);
						EXPL.DAT[side].device_size := UDINT_TO_INT(DMemInfo.memsize/1048576);
					END_IF
				END_IF

			// ----------------------------------------------------------------------------------------
			// OK
				IF ((NET.PAR.server_protocol = 'ftp' AND EXPL.PAR[side].device_active = 'NET_DEVICE') OR (DMemInfo.status = OK)) THEN
				// Select item after copy->refresh
				IF(do_select <> 0) THEN
					FOR ly:=0 TO EXPL.DAT[NOT USINT_TO_BOOL(do_select-1)].item_num DO
						IF(EXPL.DAT[USINT_TO_BOOL(do_select-1)].item_list[EXPL.VIS[USINT_TO_BOOL(do_select-1)].item_selected] = EXPL.DAT[NOT USINT_TO_BOOL(do_select-1)].item_list[ly]) THEN
							EXIT;
						END_IF
					END_FOR;
					EXPL.VIS[NOT USINT_TO_BOOL(do_select-1)].item_selected := ly;
					do_select := 0;
				END_IF
				// Reset command and return to wait state
				EXPL.CMD[side].refresh	:= FALSE;
				IF(has_oversized_items) THEN
					step := CreateError(ERR_NAME_EXCEEDS_MAX, side, step, 'one or more names exceeds maximum length', ADR(EXPL));
				ELSE
					step := EXP_WAIT;
				END_IF
				// Error
			ELSIF (DMemInfo.status <> ERR_FUB_BUSY) THEN
				step := CreateError(DMemInfo.status, side, step, 'error reading device memory information', ADR(EXPL));
			END_IF
			//**********************************************************************************************
			// Change directory
			//**********************************************************************************************
		EXP_DIR_CHANGE:
			// ----------------------------------------------------------------------------------------
			// Move one directory up
			IF (EXPL.DAT[side].item_list[EXPL.VIS[side].item_selected] = '..') THEN
				lx := brsstrlen(ADR(EXPL.PAR[side].dir_path));
				WHILE lx>0 DO
					IF(brsmemcmp(ADR(EXPL.PAR[side].dir_path) + lx, ADR('/'), 1) = 0) THEN
						EXIT;
					ELSE
						brsmemset(ADR(EXPL.PAR[side].dir_path) + lx, 0, 1);
					END_IF
					lx := lx -1;
				END_WHILE
				brsmemset(ADR(EXPL.PAR[side].dir_path) + lx, 0, 1);
				// ----------------------------------------------------------------------------------------
				// Move one directory down
			ELSE
				// Add slash if not in root
				IF(EXPL.PAR[side].dir_path <> '/') THEN
					brsstrcat(ADR(EXPL.PAR[side].dir_path), ADR('/'));
				END_IF
				brsstrcat(ADR(EXPL.PAR[side].dir_path), ADR(EXPL.DAT[side].item_list[EXPL.VIS[side].item_selected]) + 5);
				EXPL.CMD[side].refresh := 1;
			END_IF
			// Reset command and return to wait state
			EXPL.VIS[side].item_selected	:= 0;
			EXPL.CMD[side].dir_change 		:= 0;
			EXPL.CMD[side].refresh 			:= TRUE;
			step							:= EXP_WAIT;
			//**********************************************************************************************
			// Copy all items
			//**********************************************************************************************
		EXP_COPY_ALL:
			// Show current state
			animation := animation := WorkingStatus(ADR(EXPL), ADR('copying files and folders...'), animation);

			EXPL.VIS[side].item_selected := 0;
			// ----------------------------------------------------------------------------------------
			// Skip dots at the beginning of the list
			IF (EXPL.DAT[side].item_list[EXPL.VIS[side].item_selected] = '..') THEN
				EXPL.VIS[side].item_selected := EXPL.VIS[side].item_selected + 1;
			END_IF
			// Check first entry
			IF(brsmemcmp(ADR(EXPL.DAT[side].item_list[EXPL.VIS[side].item_selected]), ADR('(DIR)'), 5) = 0) THEN
				step := EXP_DIR_COPY;
			ELSE
				step := EXP_FILE_COPY;
			END_IF
			//**********************************************************************************************
			// Copy files
			//**********************************************************************************************
		EXP_FILE_COPY:
			// Show current state
			animation := WorkingStatus(ADR(EXPL), ADR('copying file...'), animation);

			// -----------------------------------------------------------------.----------------------
			// Proceed with copy all until last file is copied
			IF ((EXPL.VIS[side].item_selected < SIZEOF(EXPL.DAT[side].item_list)/SIZEOF(EXPL.DAT[side].item_list[0])) AND (EXPL.VIS[side].item_selected < EXPL.DAT[side].item_num)) THEN
				// ------------------------------------------------------------------------------------
				// Check if file name is empty
				IF (EXPL.DAT[side].item_list[EXPL.VIS[side].item_selected] <> '') THEN
					// --------------------------------------------------------------------------------
					// Check if new file name fits into string
					IF(brsstrlen(ADR(EXPL.DAT[side].item_list[EXPL.VIS[side].item_selected])) < EXPL_ITEM_LENGTH) THEN
						// ----------------------------------------------------------------------------
						// Initialize copy structure
						CreateCompletePath(EXPL.PAR[side].dir_path, EXPL.DAT[side].item_list[EXPL.VIS[side].item_selected], ADR(tmp_str3));
						CreateCompletePath(EXPL.PAR[NOT side].dir_path, EXPL.DAT[side].item_list[EXPL.VIS[side].item_selected], ADR(tmp_str4));
						FCopy.enable 	:= 1;
						FCopy.pSrcDev	:= ADR(EXPL.PAR[side].device_active);
						FCopy.pSrc		:= ADR(tmp_str3);
						FCopy.pDestDev  := ADR(EXPL.PAR[NOT side].device_active);
						FCopy.pDest		:= ADR(tmp_str4);
						FCopy.option 	:= FILE_OW_DETMEM;
						FCopy();

						// ----------------------------------------------------------------------------
						// OK
						IF (FCopy.status = OK AND EXPL.CMD[side].copy = 1) THEN
							// Select entry, reset command and refresh directory
							IF(COPY_AUTO_REFRESH = TRUE) THEN
								EXPL.CMD[NOT side].refresh := TRUE;
							END_IF
							IF(COPY_AUTO_SELECT = TRUE) THEN
								do_select := BOOL_TO_USINT(side) + 1;
							END_IF
							EXPL.CMD[side].copy	:= FALSE;
							step := EXP_WAIT;
							// ----------------------------------------------------------------------------
							// Proceed with next file
						ELSIF (FCopy.status = OK) THEN
							EXPL.VIS[side].item_selected := EXPL.VIS[side].item_selected + 1;
						ELSIF (FCopy.status <> ERR_FUB_BUSY) THEN
							step := CreateError(FCopy.status, side, step, 'error copying file', ADR(EXPL));
						END_IF
						// File name is too long
					ELSE
						step := CreateError(ERR_NAME_EXCEEDS_MAX, side, step, 'file name exceeds maximum length', ADR(EXPL));
					END_IF
					// File name  is empty
				ELSE
					step := CreateError(ERR_EMPTY_ITEM, side, step, 'file name is empty', ADR(EXPL));
				END_IF
				// ----------------------------------------------------------------------------------------
				// Finish copy all
			ELSE
				// Reset command and refresh directory
				IF(COPY_AUTO_REFRESH = TRUE) THEN
					EXPL.CMD[NOT side].refresh := TRUE;
				END_IF
				EXPL.CMD[side].copy_all			:= FALSE;
				EXPL.VIS[side].item_selected 	:= 0;
				step							:= EXP_WAIT;
			END_IF
			//**********************************************************************************************
			// Copy directory
			//**********************************************************************************************
		EXP_DIR_COPY:
			// Show current state
			animation := WorkingStatus(ADR(EXPL), ADR('copying directory...'), animation);

			// ----------------------------------------------------------------------------------------
			// Proceed with copy all until last file is copied
			IF ((EXPL.VIS[side].item_selected < SIZEOF(EXPL.DAT[side].item_list)/SIZEOF(EXPL.DAT[side].item_list[0])) AND (EXPL.VIS[side].item_selected < EXPL.DAT[side].item_num)) THEN
				IF (EXPL.DAT[side].item_list[EXPL.VIS[side].item_selected] <> '') THEN
					// --------------------------------------------------------------------------------
					// Check if new directory name fits into path string
					IF(brsstrlen(ADR(EXPL.DAT[side].item_list[EXPL.VIS[side].item_selected])) + brsstrlen(ADR(EXPL.PAR[NOT side].dir_path)) + 1 < EXPL_DIR_PATH_LENGTH) THEN
						// ----------------------------------------------------------------------------
						// Initialize copy structure
						CreateCompletePath(EXPL.PAR[side].dir_path, EXPL.DAT[side].item_list[EXPL.VIS[side].item_selected], ADR(tmp_str3));
						CreateCompletePath(EXPL.PAR[NOT side].dir_path, EXPL.DAT[side].item_list[EXPL.VIS[side].item_selected], ADR(tmp_str4));
						// ----------------------------------------------------------------------------
						// Make sure we are not copying directories recursively
						IF((EXPL.PAR[side].device_active = EXPL.PAR[NOT side].device_active) AND ((brsmemcmp(ADR(tmp_str3), ADR(tmp_str4), brsstrlen(ADR(tmp_str3))) = 0) OR (brsmemcmp(ADR(tmp_str4), ADR(tmp_str3), brsstrlen(ADR(tmp_str4))) = 0))) THEN
							step := CreateError(ERR_PATH_RECURSIVE, side, step, 'can not copy directory into itself', ADR(EXPL));
						ELSE
							DCopy.enable 	:= 1;
							DCopy.pSrcDev	:= ADR(EXPL.PAR[side].device_active);
							DCopy.pSrcDir	:= ADR(tmp_str3);
							DCopy.pDestDev 	:= ADR(EXPL.PAR[NOT side].device_active);
							DCopy.pDestDir 	:= ADR(tmp_str4);
							DCopy.option 	:= fiOVERWRITE;
							DCopy();

							// ----------------------------------------------------------------------------
							// OK
							IF (DCopy.status = OK AND EXPL.CMD[side].copy = 1) THEN
								// Reset command and refresh directory
								IF(COPY_AUTO_REFRESH = TRUE) THEN
									EXPL.CMD[NOT side].refresh := TRUE;
								END_IF
								IF (COPY_AUTO_SELECT = TRUE) THEN
									do_select := BOOL_TO_USINT(side) + 1;
								END_IF
								EXPL.CMD[side].copy	:= FALSE;
								step := EXP_WAIT;
								// ----------------------------------------------------------------------------
								// Proceed with next directory
							ELSIF (DCopy.status = OK) THEN
								EXPL.VIS[side].item_selected := EXPL.VIS[side].item_selected + 1;
								// Switch to file copy when no more directory can be found
								IF(brsmemcmp(ADR(EXPL.DAT[side].item_list[EXPL.VIS[side].item_selected]), ADR('(DIR)'), 5) <> 0) THEN
									step := EXP_FILE_COPY;
								END_IF
								// Error
							ELSIF (DCopy.status <> ERR_FUB_BUSY) THEN
								step := CreateError(DCopy.status, side, step, 'error copying directory', ADR(EXPL));
							END_IF
						END_IF
						// Directory name is too long
					ELSE
						step := CreateError(ERR_PATH_EXCEEDS_MAX, side, step, 'directory path name exceeds maximum length', ADR(EXPL));
					END_IF
					// Directory name is empty
				ELSE
					step := CreateError(ERR_EMPTY_ITEM, side, step, 'directory name is empty', ADR(EXPL));
				END_IF
				// ----------------------------------------------------------------------------------------
				// Finish copy all
			ELSE
				// Reset command and refresh directory
				IF (COPY_AUTO_REFRESH = TRUE) THEN
					EXPL.CMD[NOT side].refresh := TRUE;
				END_IF
				EXPL.CMD[side].copy_all := FALSE;
				EXPL.VIS[side].item_selected := 0;
				step := EXP_WAIT;
			END_IF
			//**********************************************************************************************
			// Delete selected file
			//**********************************************************************************************
		EXP_FILE_DELETE:
			// Show current state
			animation := WorkingStatus(ADR(EXPL), ADR('deleting file...'), animation);

			// ----------------------------------------------------------------------------------------
			// Initialize file delete structure
			CreateCompletePath(EXPL.PAR[side].dir_path, item_name, ADR(tmp_str3));
			FDelete.enable		:= TRUE;
			FDelete.pDevice 	:= ADR(EXPL.PAR[side].device_active);
			FDelete.pName		:= ADR(tmp_str3);
			FDelete();

			// ----------------------------------------------------------------------------------------
			// OK
			IF (FDelete.status = OK) THEN
				// Reset command delete and return to wait state
				IF(EXPL.CMD[side].delete = TRUE) THEN
					EXPL.CMD[side].delete 	:= FALSE;
					EXPL.CMD[side].refresh  := TRUE;
					step := EXP_WAIT;
					// Proceed with command upload
				ELSE
					step := EXP_FILE_UPLOAD_1;
				END_IF
				// Error
			ELSIF (FDelete.status <> ERR_FUB_BUSY) THEN
				step := CreateError(FDelete.status, side, step, 'error deleting file', ADR(EXPL));
			END_IF
			//**********************************************************************************************
			// Rename selected file
			//**********************************************************************************************
		EXP_FILE_RENAME:
			// Show current state
			animation := WorkingStatus(ADR(EXPL), ADR('renaming file...'), animation);

			// ----------------------------------------------------------------------------------------
			// Initialize file delete structure
			CreateCompletePath(EXPL.PAR[side].dir_path, EXPL.DAT[side].item_list[EXPL.VIS[side].item_selected], ADR(tmp_str2));
			CreateCompletePath(EXPL.PAR[side].dir_path, EXPL.PAR[side].new_name, ADR(tmp_str3));
			FRename.enable		:= TRUE;
			FRename.pDevice 	:= ADR(EXPL.PAR[side].device_active);
			FRename.pName		:= ADR(tmp_str2);
			FRename.pNewName	:= ADR(tmp_str3);
			FRename();

			// ----------------------------------------------------------------------------------------
			// OK
			IF (FRename.status = OK) THEN
				// Reset command and return to wait state
				EXPL.CMD[side].rename 	:= FALSE;
				EXPL.CMD[side].refresh  := TRUE;
				step := EXP_WAIT;
				// Error
			ELSIF (FRename.status <> ERR_FUB_BUSY) THEN
				step := CreateError(FRename.status, side, step, 'error renaming file', ADR(EXPL));
			END_IF
			//**********************************************************************************************
			// Duplicate selected file
			//**********************************************************************************************
		EXP_FILE_DUPLICATE:
			// Show current state
			animation := WorkingStatus(ADR(EXPL), ADR('duplicating file...'), animation);

			// Build automatic name "<name>_<index>.<ext>" when no custom name is given
			IF (EXPL.PAR[side].new_name = '') THEN
				IF (duplicate_index = 0) THEN
					duplicate_index := 1;
					brsmemset(ADR(duplicate_base_name), 0, SIZEOF(duplicate_base_name));
					brsmemset(ADR(duplicate_extension), 0, SIZEOF(duplicate_extension));
					brsmemset(ADR(duplicate_suffix_text), 0, SIZEOF(duplicate_suffix_text));
					duplicate_dot_pos := FindInMem(ADR(item_name), brsstrlen(ADR(item_name)), ADR('.'), 1, TRUE);
					IF (duplicate_dot_pos > 0) THEN
						brsmemcpy(ADR(duplicate_base_name), ADR(item_name), DINT_TO_UDINT(duplicate_dot_pos));
						brsstrcpy(ADR(duplicate_extension), ADR(item_name) + DINT_TO_UDINT(duplicate_dot_pos));
					ELSE
						brsstrcpy(ADR(duplicate_base_name), ADR(item_name));
					END_IF

					// If base name ends with _<number>, continue counting from that number.
					duplicate_suffix_pos := FindInMem(ADR(duplicate_base_name), brsstrlen(ADR(duplicate_base_name)), ADR('_'), 1, TRUE);
					IF (duplicate_suffix_pos > 0 AND duplicate_suffix_pos < DINT_TO_UDINT(brsstrlen(ADR(duplicate_base_name))) - 1) THEN
						brsstrcpy(ADR(duplicate_suffix_text), ADR(duplicate_base_name) + DINT_TO_UDINT(duplicate_suffix_pos + 1));
						duplicate_suffix_valid := TRUE;
						FOR lx := 0 TO brsstrlen(ADR(duplicate_suffix_text)) - 1 DO
							IF (brsmemcmp(ADR(duplicate_suffix_text) + lx, ADR('0'), 1) < 0 OR brsmemcmp(ADR(duplicate_suffix_text) + lx, ADR('9'), 1) > 0) THEN
								duplicate_suffix_valid := FALSE;
								EXIT;
							END_IF
						END_FOR

						IF (duplicate_suffix_valid) THEN
							duplicate_index := DINT_TO_UDINT(brsatoi(ADR(duplicate_suffix_text)) + 1);
							brsmemset(ADR(duplicate_base_name) + DINT_TO_UDINT(duplicate_suffix_pos), 0, 1);
						END_IF
					END_IF
				END_IF

				brsmemset(ADR(tmp_str2), 0, SIZEOF(tmp_str2));
				brsmemset(ADR(tmp_str4), 0, SIZEOF(tmp_str4));
				brsstrcpy(ADR(tmp_str4), ADR(duplicate_base_name));
				brsstrcat(ADR(tmp_str4), ADR('_'));
				brsitoa(UDINT_TO_DINT(duplicate_index), ADR(tmp_str2));
				brsstrcat(ADR(tmp_str4), ADR(tmp_str2));
				brsstrcat(ADR(tmp_str4), ADR(duplicate_extension));
			ELSE
				brsstrcpy(ADR(tmp_str4), ADR(EXPL.PAR[side].new_name));
			END_IF

			// Verify final name and path length before calling FileCopy
			IF (brsstrlen(ADR(tmp_str4)) = 0) THEN
				step := CreateError(ERR_EMPTY_ITEM, side, step, 'duplicate target name is empty', ADR(EXPL));
			ELSIF (brsstrlen(ADR(tmp_str4)) >= EXPL_ITEM_LENGTH) THEN
				step := CreateError(ERR_NAME_EXCEEDS_MAX, side, step, 'duplicate file name exceeds maximum length', ADR(EXPL));
			ELSIF (brsstrlen(ADR(tmp_str4)) + brsstrlen(ADR(EXPL.PAR[side].dir_path)) + 1 >= EXPL_DIR_PATH_LENGTH) THEN
				step := CreateError(ERR_PATH_EXCEEDS_MAX, side, step, 'duplicate file path exceeds maximum length', ADR(EXPL));
			ELSE
				CreateCompletePath(EXPL.PAR[side].dir_path, item_name, ADR(tmp_str2));
				CreateCompletePath(EXPL.PAR[side].dir_path, tmp_str4, ADR(tmp_str3));

				FCopy.enable 	:= TRUE;
				FCopy.pSrcDev	:= ADR(EXPL.PAR[side].device_active);
				FCopy.pSrc		:= ADR(tmp_str2);
				FCopy.pDestDev := ADR(EXPL.PAR[side].device_active);
				FCopy.pDest		:= ADR(tmp_str3);
				FCopy.option 	:= 0;
				FCopy();

				IF (FCopy.status = OK) THEN
					EXPL.CMD[side].duplicate := FALSE;
					EXPL.CMD[side].refresh := TRUE;
					step := EXP_WAIT;
				ELSIF (FCopy.status = fiERR_EXIST AND EXPL.PAR[side].new_name = '') THEN
					duplicate_index := duplicate_index + 1;
				ELSIF (FCopy.status <> ERR_FUB_BUSY) THEN
					step := CreateError(FCopy.status, side, step, 'error duplicating file', ADR(EXPL));
				END_IF
			END_IF
			//**********************************************************************************************
			// View selected file
			//**********************************************************************************************
		EXP_FILE_VIEW:
			CreateCompletePath(EXPL.PAR[side].dir_path, EXPL.DAT[side].item_list[EXPL.VIS[side].item_selected], ADR(tmp_str1));

			FOR lx:=0 TO SIZEOF(EXPL_VIEW_FILTER)/SIZEOF(EXPL_VIEW_FILTER[0]) - 1 DO
				IF(brsstrlen(ADR(tmp_str1)) >= brsstrlen(ADR(EXPL_VIEW_FILTER[lx])) AND EXPL_VIEW_FILTER[lx] <> '') THEN
					// --------------------------------------------------------------------------------
					// Verify that file name contains filter
					IF(brsmemcmp(ADR(tmp_str1) + brsstrlen(ADR(tmp_str1)) - brsstrlen(ADR(EXPL_VIEW_FILTER[lx])) , ADR(EXPL_VIEW_FILTER[lx]), brsstrlen(ADR(EXPL_VIEW_FILTER[lx]))) = 0) THEN
						EXPL.VIS[side].view_file_path := '/FileDevice:';
						brsstrcat(ADR(EXPL.VIS[side].view_file_path), ADR(EXPL.PAR[side].device_active));
						IF(brsmemcmp(ADR(tmp_str1), ADR('/'), 1) <> 0) THEN
							brsstrcat(ADR(EXPL.VIS[side].view_file_path), ADR('/'));
						END_IF
						brsstrcat(ADR(EXPL.VIS[side].view_file_path), ADR(tmp_str1));
						EXPL.CMD[side].view_file := FALSE;
						EXPL.VIS[side].view_file := TRUE;
						step := EXP_WAIT;
						RETURN;
					END_IF
				END_IF
			END_FOR;
			step := CreateError(FRename.status, side, step, 'error this file extension is not supported for viewing', ADR(EXPL));
			//**********************************************************************************************
			// Download file
			//**********************************************************************************************
		EXP_FILE_DOWNLOAD:
			animation := WorkingStatus(ADR(EXPL), ADR('downloading file...'), animation);

			EXPL.VIS[side].file_full_path := device_active;
			IF dir_path <> '' THEN
				brsstrcat(ADR(EXPL.VIS[side].file_full_path), ADR(dir_path));
			END_IF
			brsstrcat(ADR(EXPL.VIS[side].file_full_path), ADR('/'));
			brsstrcat(ADR(EXPL.VIS[side].file_full_path), ADR(item_name));

			EXPL.VIS[side].file_status := 0;
			EXPL.VIS[side].download_execute := TRUE;
			step := EXP_FILE_DOWNLOAD_1;

			//**********************************************************************************************
			// Download file
			//**********************************************************************************************
		EXP_FILE_DOWNLOAD_1:
			IF EDGENEG(EXPL.VIS[side].download_execute) THEN
				EXPL.CMD[side].download := FALSE;

				// ----------------------------------------------------------------------------------------
				// OK
				IF (EXPL.VIS[side].file_status = OK) THEN
					step := EXP_WAIT;
					// Error access rights
				ELSIF (EXPL.VIS[side].file_status = -1064165358) THEN
					step := CreateError(EXPL.VIS[side].file_status, side, step, 'user  has insufficient rights to access file or device', ADR(EXPL));
					// Error
				ELSE
					step := CreateError(EXPL.VIS[side].file_status, side, step, 'error downloading file', ADR(EXPL));
				END_IF
			END_IF
			//**********************************************************************************************
			// Download all files
			//**********************************************************************************************
		EXP_FILE_DOWNLOAD_DIR:
			// Show current state
			animation := WorkingStatus(ADR(EXPL), ADR('processing directory...'), animation);
			tmp_str1 := item_name;
			brsstrcat(ADR(tmp_str1), ADR('.tar.gz'));

			// ----------------------------------------------------------------------------------------
			// Initialize file zip structure
			CreateCompletePath(EXPL.PAR[side].dir_path, EXPL.DAT[side].item_list[EXPL.VIS[side].item_selected], ADR(tmp_str2));

			zipArchive_0.enable := 1;
			zipArchive_0.pArchiveDevice := ADR('TMP_USER');
			zipArchive_0.pArchiveFile := ADR(tmp_str1);
			zipArchive_0.pSrcDevice := ADR(EXPL.PAR[side].device_active);
			zipArchive_0.pSrcFile := ADR(tmp_str2);
			zipArchive_0.pOptions := ADR('/COMPRESSION_LEVEL=7');
			zipArchive_0();

			// ----------------------------------------------------------------------------------------
			// OK
			IF (zipArchive_0.status = OK) THEN
				item_name := tmp_str1;
				device_active := 'TMP_USER';
				dir_path := '';
				step := EXP_FILE_DOWNLOAD;
				// Error
			ELSIF (zipArchive_0.status <> ERR_FUB_BUSY) THEN
				step := CreateError(zipArchive_0.status, side, step, 'error creating zip file', ADR(EXPL));
			END_IF
			//**********************************************************************************************
			// Upload file - verify parameters
			//**********************************************************************************************
		EXP_FILE_UPLOAD:
			// Show current state
			animation := WorkingStatus(ADR(EXPL), ADR('uploading file...'), animation);

			EXPL.VIS[side].file_full_path := device_active;
			brsstrcat(ADR(EXPL.VIS[side].file_full_path), ADR(dir_path));
			brsstrcat(ADR(EXPL.VIS[side].file_full_path), ADR('/'));

			EXPL.VIS[side].file_status := 0;
			EXPL.VIS[side].upload_execute := TRUE;
			step := EXP_FILE_UPLOAD_1;

			//**********************************************************************************************
			// Upload file
			//**********************************************************************************************
		EXP_FILE_UPLOAD_1:
			IF (EXPL.VIS[side].upload_execute = FALSE) THEN
				EXPL.CMD[side].upload := FALSE;

				// ----------------------------------------------------------------------------------------
				// OK
				IF (EXPL.VIS[side].file_status = OK) THEN
					EXPL.CMD[side].refresh := 1;

					step := EXP_WAIT;
				// Error file name length
				ELSIF (EXPL.VIS[side].file_status = 10103) THEN
					step := CreateError(EXPL.VIS[side].file_status, side, step, 'file name exceeds maximum length', ADR(EXPL));
				// Error file size
				ELSIF (EXPL.VIS[side].file_status = 10101) THEN
					step := CreateError(EXPL.VIS[side].file_status, side, step, 'maximum file size exceeded', ADR(EXPL));
				// Error access rights
				ELSIF (EXPL.VIS[side].file_status = -1064165358) THEN
					step := CreateError(EXPL.VIS[side].file_status, side, step, 'user  has insufficient rights to access file or device', ADR(EXPL));
				// Error
				ELSE
					step := CreateError(EXPL.VIS[side].file_status, side, step, 'error uploading file', ADR(EXPL));
				END_IF
			END_IF

			//**********************************************************************************************
			// Create new directory
			//**********************************************************************************************
		EXP_DIR_CREATE:
			// Show current state
			animation := WorkingStatus(ADR(EXPL), ADR('creating directory...'), animation);

			// ----------------------------------------------------------------------------------------
			// Initialize directory create structure
			CreateCompletePath(EXPL.PAR[side].dir_path, EXPL.PAR[side].new_name, ADR(tmp_str3));
			DCreate.enable	:= 1;
			DCreate.pDevice := ADR(EXPL.PAR[side].device_active);
			DCreate.pName 	:= ADR(tmp_str3);
			DCreate();

			// ----------------------------------------------------------------------------------------
			// OK
			IF (DCreate.status = OK) THEN
				// Reset command and return to wait state
				EXPL.CMD[side].dir_create 	:= FALSE;
				EXPL.CMD[side].refresh 		:= TRUE;
				step := EXP_WAIT;
				// Error
			ELSIF (DCreate.status <> ERR_FUB_BUSY) THEN
				step := CreateError(DCreate.status, side, step, 'error creating directory', ADR(EXPL));
			END_IF
			//**********************************************************************************************
			// Delete selected directory
			//**********************************************************************************************
		EXP_DIR_DELETE:
			// Show current state
			animation := WorkingStatus(ADR(EXPL), ADR('deleting directory...'), animation);

			// ----------------------------------------------------------------------------------------
			// Initialize directory delete structure
			CreateCompletePath(EXPL.PAR[side].dir_path, item_name, ADR(tmp_str3));
			DDelete.enable	:= TRUE;
			DDelete.pDevice := ADR(EXPL.PAR[side].device_active);
			DDelete.pName 	:= ADR(tmp_str3);
			DDelete();

			// ----------------------------------------------------------------------------------------
			// OK
			IF (DDelete.status = OK) THEN
				// Reset command and return to wait state
				EXPL.CMD[side].delete := FALSE;
				EXPL.CMD[side].refresh := TRUE;
				step := EXP_WAIT;
				// Error
			ELSIF (DDelete.status <> ERR_FUB_BUSY) THEN
				step := CreateError(DDelete.status, side, step, 'error deleting directory', ADR(EXPL));
			END_IF
			//**********************************************************************************************
			// Rename selected directory
			//**********************************************************************************************
		EXP_DIR_RENAME:
			// Show current state
			animation := WorkingStatus(ADR(EXPL), ADR('renaming directory...'), animation);

			// ----------------------------------------------------------------------------------------
			// Initialize file delete structure
			CreateCompletePath(EXPL.PAR[side].dir_path, EXPL.DAT[side].item_list[EXPL.VIS[side].item_selected], ADR(tmp_str2));
			CreateCompletePath(EXPL.PAR[side].dir_path, EXPL.PAR[side].new_name, ADR(tmp_str3));
			DRename.enable		:= TRUE;
			DRename.pDevice 	:= ADR(EXPL.PAR[side].device_active);
			DRename.pName		:= ADR(tmp_str2);
			DRename.pNewName	:= ADR(tmp_str3);
			DRename();

			// ----------------------------------------------------------------------------------------
			// OK
			IF (DRename.status = OK) THEN
				// Reset command and return to wait state
				EXPL.CMD[side].rename 	:= FALSE;
				EXPL.CMD[side].refresh  := TRUE;
				step := EXP_WAIT;
				// Error
			ELSIF (DRename.status <> ERR_FUB_BUSY) THEN
				step := CreateError(DRename.status, side, step, 'error renaming directory', ADR(EXPL));
			END_IF
			//**********************************************************************************************
			// Overwrite file - Check if file exists
			//**********************************************************************************************
		EXP_OVERWRITE_1:
			EXPL.VIS[side].overwrite_response := NONE;

			// ----------------------------------------------------------------------------------------
			// Checking for files with the same name
			FOR lx:=0 TO EXPL.DAT[side].item_num DO
				IF(EXPL.CMD[side].copy = TRUE AND EXPL.DAT[NOT side].item_list[lx] = item_name) THEN
					EXPL.VIS[side].overwrite_request := TRUE;
					step := EXP_OVERWRITE_2;
					RETURN;
				END_IF;
			END_FOR;

			// Proceed with copy command
			IF(brsmemcmp(ADR(item_name), ADR('(DIR)'), 5) = 0)	THEN
				step := EXP_DIR_COPY;
			ELSE
				step := EXP_FILE_COPY;
			END_IF
			//**********************************************************************************************
			// Overwrite file - Wait for message box response
			//**********************************************************************************************
		EXP_OVERWRITE_2:
			// Overwrite file
			IF(EXPL.VIS[side].overwrite_response = YES) THEN
				// Proceed with copy command
				IF(brsmemcmp(ADR(item_name), ADR('(DIR)'), 5) = 0)	THEN
					step := EXP_DIR_COPY;
				ELSE
					step := EXP_FILE_COPY;
				END_IF
				EXPL.VIS[side].overwrite_request := FALSE;

			// Do not overwrite file
			ELSIF(EXPL.VIS[side].overwrite_response = NO) THEN
				// Reset copy command
				EXPL.CMD[side].copy	:= FALSE;
				EXPL.VIS[side].overwrite_request := FALSE;
				step := EXP_WAIT;
			END_IF
	END_CASE

END_PROGRAM
```

### changelog.txt
```
04.09.2026
- Fixed FTP root file operations by using relative paths without a leading slash
- Skip device memory information for FTP network devices
- Fixed the mappView root file URL separator after relative path generation
- Added protocol-specific network device parameters and an option to ignore ping failures
- Removed the SYSTEM entry from the predefined device list

27.04.2026
- Added new command duplicate
- Check file name length during command rename and upload

07.01.2026
- Better error message when upload file size exceeds maximum

Version 2.0
- Update to Automation Studio AS 6.3 and mapp 6.4
- Replaced upload and download with transfer widget

Version 1.9
- Update to Automation Studio AS 4.12 and mapp 5.24

Version 1.8
- Update to Automation Studio AS 4.9 and runtime D4.90
- Revert fix from build 1.7 since bug in AsHTTP is fixed in D4.90

Version 1.7
- Fixed data start offset in upload was not correct
- Fixed upload file name can exceed EXPL_ITEM_LENGTH
- Fixed upload crashing CPU when it exceeds EXPL_UPLOAD_DOWNLOAD_SIZE

Version 1.6
- Fixed reset button was disabled for network and USB
- Fixed network root directory is showing all as directories
- Fixed copy directory does not report error
- Added ping OK button to network share configuration page
- Network can now be disconnected with the Reset / Abort button

Version 1.5
- Update USB helper task
- Update NET helper task
- Prevent user from copying directories recursively

Version 1.4
- Added support for folder download
- Renamed status to status_text and added status_no to show busy state and error numbers

Version 1.3
- Code cleanup
- UI Tweaks
- Added file device memory information
- Added current directory entry to be compatible with network shares
- Change from static IP to DHCP
- Fixed filter text field and button is disabled when no files are visible
- Fixed file size calculation
- Fixed ReplaceString function call
- Fixed error is not showing up in wait state
- Fixed dir read and file write error is not reported

Version 1.2
- Fixed download not working when downloading the same file again
- Fixed upload not working with large files > 1 MB

Version 1.1
- Fixed file open click event
- Added support multiple USB sticks
- Added message box when uploading or copying file that exists on target
- Fixed button rename is not disabled when command is running

Version 1.0
- Added support for file download over mappView
- Added support for file upload over mappView
- Code cleanup

Version 0.9
- Added function to view files by double click or command

Version 0.8
- Added function for generating list box data provider
- Fixed typos, cleaned up binding file
- Created individual packages for NET and USB
- Fixed enable/disable
- Added message box before deleting an item

Version 0.7
- New function rename file or folder
- Fixed memory leak when last entry in list is used
- Code optimizations

Version 0.6
- Changed upper limit of USB polling interval
- Removed obsolete error numbers
- Replaced error numbers with constants
- Removed obsolete variables
- Fixed old_filter variable size
- Fixed file size added to file name
- Disable file device and filter during operation

Version 0.5
- Main task ported to structure text
- Allow oversized names for files and folders
- Fixed variables types
- Applied python naming convention to all code

Version 0.2
- Added configuration for network connections
- Code cleanup

Version 0.1
- First public release
```

### NetTypes.typ
```iecst
TYPE
	netSTATE :
		(
		NET_WAIT, (*Function step: Wait for starting the Function chain*)
		NET_LINK_DEVICE, (*Function step: Link file device*)
		NET_UNLINK_DEVICE, (*Function step: Unlink the File Device from specific path*)
		NET_ERROR (*Function step: Jump to this step in every case of Error occuring in the Function chain*)
		);
	netCMD : 	STRUCT
		connect : BOOL; (*Connect to network share*)
		disconnect : BOOL; (*Disconnect from network share*)
		error_reset : BOOL; (*Reset error*)
	END_STRUCT;
	netPAR : 	STRUCT
		server_name : STRING[80]; (*Use server name*)
		server_ip : STRING[80] := '192.168.0.10'; (*or IP address*)
		server_port : STRING[80]; (*Uses default port when empty*)
		server_protocol : STRING[80] := 'cifs'; (*Type of network connection*)
		server_domain : STRING[80]; (*Domain name*)
		server_share : STRING[80] := 'share'; (*Name of the shared folder*)
		user_name : STRING[80] := 'user'; (*User name*)
		user_password : STRING[80] := 'password'; (*User password*)
		ignore_ping : BOOL := FALSE; (*Ignore ping and do not auto disconnect*)
		enable_connect : BOOL; (*Enable button connect*)
		can_ping : BOOL; (*Indicates that the network share can be pinged*)
		is_linked : BOOL; (*Network share is connected*)
	END_STRUCT;
	netERR : 	STRUCT
		state : netSTATE;
		text : STRING[80]; (*Error text*)
	END_STRUCT;
	netMAIN : 	STRUCT
		CMD : netCMD; (*Command structure*)
		PAR : netPAR; (*Parameter structure*)
		ERR : netERR; (*Error structure*)
		status : UINT;
	END_STRUCT;
END_TYPE
```

### Program Logical/NETdevice/NetDevice

#### Main.st
```iecst
PROGRAM _INIT
END_PROGRAM

PROGRAM _CYCLIC
	// Trigger ping request
	IF NOT NET.PAR.ignore_ping THEN
		PingTimer.IN := TRUE;
		PingTimer.PT := PING_TIMEOUT;
		PingTimer();
		// Try to ping network share if not connected
		IF((NET.PAR.server_ip <> '' OR NET.PAR.server_name <> '') AND PingTimer.Q) THEN
			// Use IPÜ address
			IF(NET.PAR.server_ip <> '') THEN
				IcmpPing_0(enable := TRUE, pHost := ADR(NET.PAR.server_ip), timeout := PING_TIMEOUT);
			// Use host name
			ELSE
				IcmpPing_0(enable := TRUE, pHost := ADR(NET.PAR.server_name), timeout := PING_TIMEOUT);
			END_IF
			// Ping was OK
			IF(IcmpPing_0.status = ERR_OK) THEN
				PingTimer(IN := FALSE);
				NET.PAR.can_ping := TRUE;
			// Disconnect from share when ping failed
			ELSIF(IcmpPing_0.status <> ERR_FUB_BUSY) THEN
				PingTimer(IN := FALSE);
				NET.PAR.can_ping := FALSE;
				IF(NET.PAR.is_linked) THEN
					NET.CMD.disconnect := TRUE;
				END_IF
			END_IF
		ELSIF(PingTimer.Q) THEN
			PingTimer(IN := FALSE);
		END_IF
	END_IF

	CASE state_machine OF
		// -----------------------------------------------------------------------------------------------------------
		// Wait state
		// -----------------------------------------------------------------------------------------------------------
		NET_WAIT:
			NET.PAR.enable_connect := TRUE;
			NET.status := ERR_OK;
			// --------------------------------------------------------------------------------------------------------------------
			// Connect to server
			IF(NET.CMD.connect) THEN
				DevLink_0(enable := FALSE);
				IF(NET.PAR.is_linked) THEN
					state_machine := NET_UNLINK_DEVICE;
				ELSE
					state_machine := NET_LINK_DEVICE;
				END_IF
				NET.status := ERR_FUB_BUSY;
			END_IF
			// --------------------------------------------------------------------------------------------------------------------
			// Disconnect from server
			IF(NET.CMD.disconnect) THEN
				DevUnlink_0.enable := FALSE;
				DevUnlink_0;
				state_machine := NET_UNLINK_DEVICE;
			END_IF
			// --------------------------------------------------------------------------------------------------------------------
			// Reset error
			IF(NET.CMD.error_reset) THEN
				NET.CMD.error_reset := FALSE;
				brsmemset(ADR(NET.ERR), 0, SIZEOF(NET.ERR));
			END_IF
		// -----------------------------------------------------------------------------------------------------------
		// Link device
		// -----------------------------------------------------------------------------------------------------------
		NET_LINK_DEVICE:
			// Create device string
			NET.PAR.enable_connect := FALSE;
			brsmemset(ADR(device_param), 0, SIZEOF(device_param));
			IF(brsstrcmp(ADR(NET.PAR.server_name), ADR('')) <> 0) THEN
				brsstrcat(ADR(device_param), ADR('/SNAME='));
				brsstrcat(ADR(device_param), ADR(NET.PAR.server_name));
				brsstrcat(ADR(device_param), ADR(' '));
			END_IF
			IF(brsstrcmp(ADR(NET.PAR.server_ip), ADR('')) <> 0) THEN
				brsstrcat(ADR(device_param), ADR('/SIP='));
				brsstrcat(ADR(device_param), ADR(NET.PAR.server_ip));
				brsstrcat(ADR(device_param), ADR(' '));
			END_IF
			IF(brsstrcmp(ADR(NET.PAR.server_protocol), ADR('')) <> 0) THEN
				brsstrcat(ADR(device_param), ADR('/PROTOCOL='));
				brsstrcat(ADR(device_param), ADR(NET.PAR.server_protocol));
				brsstrcat(ADR(device_param), ADR(' '));
			END_IF
			IF(brsstrcmp(ADR(NET.PAR.server_protocol), ADR('tftp')) = 0) THEN
				IF(brsstrcmp(ADR(NET.PAR.server_port), ADR('')) <> 0) THEN
					brsstrcat(ADR(device_param), ADR('/PORT='));
					brsstrcat(ADR(device_param), ADR(NET.PAR.server_port));
					brsstrcat(ADR(device_param), ADR(' '));
				END_IF
			END_IF
			IF(brsstrcmp(ADR(NET.PAR.server_protocol), ADR('cifs')) = 0) THEN
				IF(brsstrcmp(ADR(NET.PAR.server_domain), ADR('')) <> 0) THEN
					brsstrcat(ADR(device_param), ADR('/DOMAIN='));
					brsstrcat(ADR(device_param), ADR(NET.PAR.server_domain));
					brsstrcat(ADR(device_param), ADR(' '));
				END_IF
				IF(brsstrcmp(ADR(NET.PAR.server_share), ADR('')) <> 0) THEN
					brsstrcat(ADR(device_param), ADR('/SHARE='));
					brsstrcat(ADR(device_param), ADR(NET.PAR.server_share));
					brsstrcat(ADR(device_param), ADR(' '));
				END_IF
			END_IF
			IF(brsstrcmp(ADR(NET.PAR.user_name), ADR('')) <> 0) THEN
				brsstrcat(ADR(device_param), ADR('/USER='));
				brsstrcat(ADR(device_param), ADR(NET.PAR.user_name));
				brsstrcat(ADR(device_param), ADR(' '));
			END_IF
			IF(brsstrcmp(ADR(NET.PAR.user_password), ADR('')) <> 0) THEN
				brsstrcat(ADR(device_param), ADR('/PASSWORD='));
				brsstrcat(ADR(device_param), ADR(NET.PAR.user_password));
				brsstrcat(ADR(device_param), ADR(' '));
			END_IF

			// Link device
			DevLink_0.enable := TRUE;
			DevLink_0.pDevice := ADR('NET_DEVICE');
			DevLink_0.pParam := ADR(device_param);
			DevLink_0;

			// --------------------------------------------------------------------------------------------------------------------
			// Success
			IF DevLink_0.status = 0 THEN
				NET.PAR.is_linked := TRUE;
				NET.CMD.connect := FALSE;
				state_machine := NET_WAIT;
			// --------------------------------------------------------------------------------------------------------------------
			// Abort command
			ELSIF(NET.CMD.error_reset = TRUE OR NET.CMD.disconnect = TRUE) THEN
				IF(DevLink_0.handle = 0) THEN
					DevLink_0(enable := FALSE);
					brsmemset(ADR(NET.CMD), 0, SIZEOF(NET.CMD));
					state_machine := NET_WAIT;
				ELSE
					state_machine := NET_UNLINK_DEVICE;
				END_IF
			// Error
			ELSIF DevLink_0.status <> ERR_FUB_BUSY THEN
				NET.ERR.state := state_machine;
				NET.ERR.text := 'error linking device';
				NET.status := DevLink_0.status;
				state_machine := NET_ERROR;
			END_IF;
		// -----------------------------------------------------------------------------------------------------------
		// UnLink device
		// -----------------------------------------------------------------------------------------------------------
		NET_UNLINK_DEVICE:
			NET.PAR.enable_connect := FALSE;
			DevUnlink_0.enable := TRUE;
			DevUnlink_0.handle := DevLink_0.handle;
			DevUnlink_0;

			// --------------------------------------------------------------------------------------------------------------------
			// Success
			IF DevUnlink_0.status = 0 THEN
				brsmemset(ADR(NET.CMD), 0, SIZEOF(NET.CMD));
				NET.PAR.is_linked := FALSE;
				DevLink_0(enable := FALSE);
				IF(NET.CMD.connect) THEN
					state_machine := NET_LINK_DEVICE;
				ELSE
					state_machine := NET_WAIT;
				END_IF
			// Error
			ELSIF DevUnlink_0.status <> ERR_FUB_BUSY THEN
				NET.CMD.error_reset := FALSE;
				NET.ERR.state := state_machine;
				NET.ERR.text := 'error unlinking device';
				NET.status := DevUnlink_0.status;
				state_machine := NET_ERROR;
			END_IF;
		// -----------------------------------------------------------------------------------------------------------
		// Error step
		// -----------------------------------------------------------------------------------------------------------
		NET_ERROR:
			// Reset commands
			NET.PAR.enable_connect := FALSE;
			NET.CMD.connect := FALSE;
			NET.CMD.disconnect := FALSE;

			// Get more error information
			IF(NET.status = 0) THEN
				NET.status := FileIoGetSysError();
			END_IF
			IF(NET.status = 26228) THEN
				brsstrcpy(ADR(NET.ERR.text), ADR('connection rejected: check network protocol, username and password'));
			ELSIF(DevLink_0.status = fiERR_DEVICE_ALREADY_EXIST) THEN
				brsstrcpy(ADR(NET.ERR.text), ADR('device is already connected'));
			END_IF

			// Reset error
			IF(NET.CMD.error_reset) THEN
				NET.CMD.error_reset := FALSE;
				brsmemset(ADR(NET.ERR), 0, SIZEOF(NET.ERR));
				DevLink_0(enable := FALSE);
				DevUnlink_0(enable := FALSE);
				state_machine := NET_WAIT;
			END_IF
	END_CASE;

END_PROGRAM

PROGRAM _EXIT
	REPEAT
		DevUnlink_0.enable := TRUE;
		DevUnlink_0.handle := DevLink_0.handle;
		DevUnlink_0;
		UNTIL DevUnlink_0.status <> ERR_FUB_BUSY
	END_REPEAT;
END_PROGRAM
```

### Program Logical/USBdevice/UsbDevice
